FUNCTION F_ContactorControl
VAR_IN_OUT
	bCtrltimerQ: BOOL;
END_VAR
VAR
END_VAR
VAR_OUTPUT
END_VAR

IF bCtrltimerQ = 0 THEN
	IO.reactorTemperatureContactor := 1;
ELSE
	IO.reactorTemperatureContactor := 0;
END_IF

END_FUNCTION

(* stored: Version 1.1.0.1, ProductVersion 3.1.4024.9
   POU F_ContactorControl: Id {070fb794-3a32-4334-af96-757ec4b76403}, SpecialFunc None *)
